// TIA Portal V20 export
TYPE "LER_typeStep"
// stored: Access Published
   STRUCT
      action { ExternalWritable := 'False'} : Array[0..9999] of Bool;
      transition { ExternalWritable := 'False'} : Array[0..9999] of Bool;
   END_STRUCT;
END_TYPE
